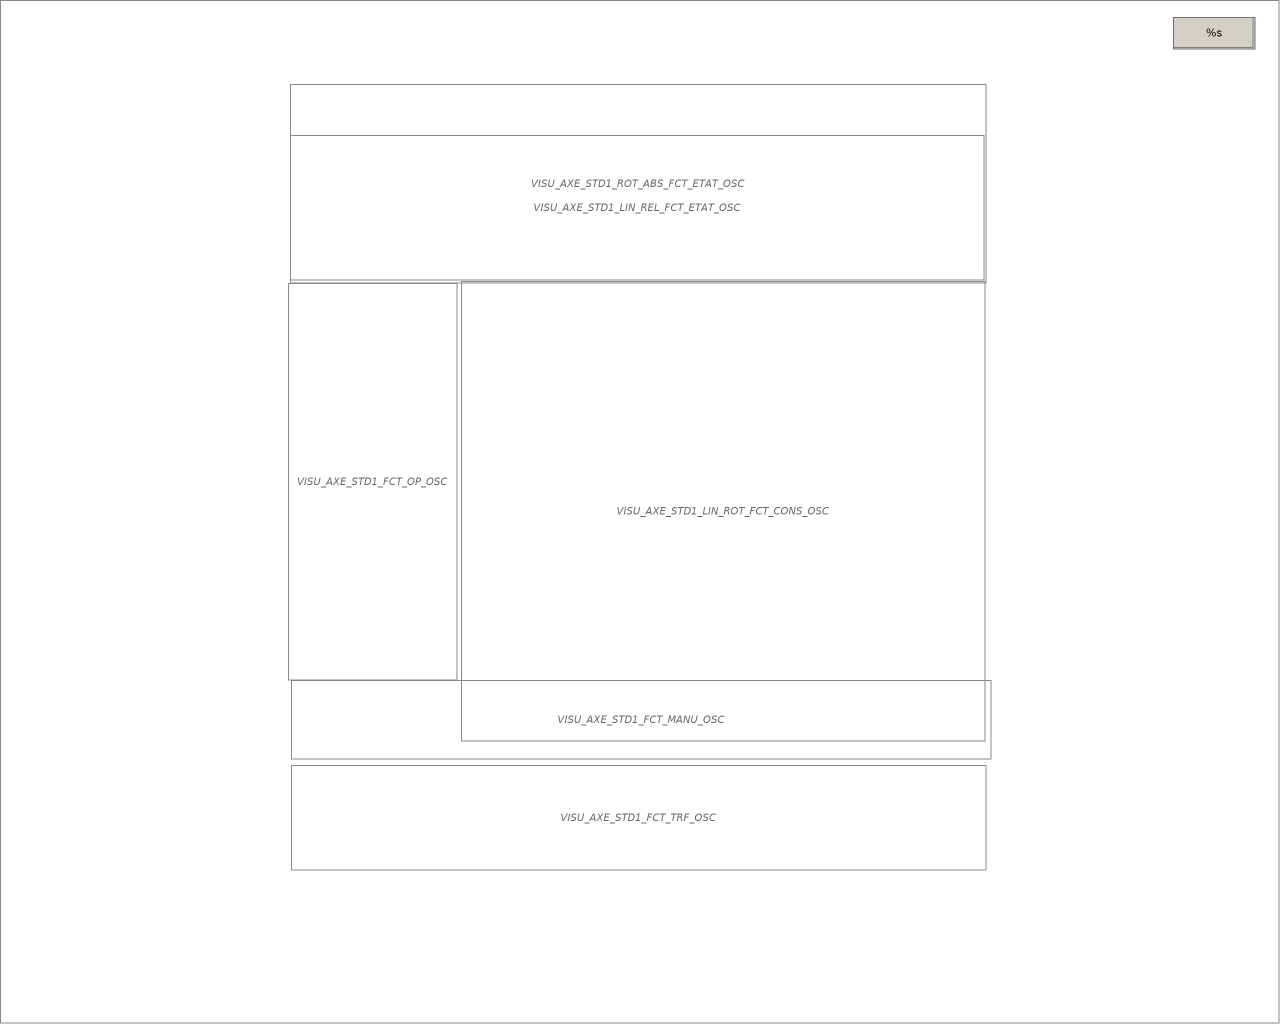
VISUALIZATION VISU_AXE_STD1_MANU_OSC  // 1280x1024
VAR_IN_OUT
	m_Input_MOTEUR: BLOCK_AXE_STD1_OSCILLANT;
	m_Input_PRG_MOUVEMENT_PS: BLOCK_PRG_MOUVEMENT_PS;
END_VAR
VAR_INPUT
	m_Input_ID_NOM_XML : INT;
	m_Input_INDEX_MOTEUR : INT;
	m_Input_Ref_Trf:	USINT;
END_VAR
    Frame (290,84 696x199), invisible if: NOT m_Input_PRG_MOUVEMENT_PS.CONF_ROT_ABS[m_Input_INDEX_MOTEUR]
        shows VISU_AXE_STD1_ROT_ABS_FCT_ETAT_OSC(m_Input_MOTEUR := m_Input_MOTEUR, m_Input_PRG_MOUVEMENT_PS := m_Input_PRG_MOUVEMENT_PS, m_Input_ID_NOM_XML := m_Input_ID_NOM_XML, m_Input_INDEX_MOTEUR := m_Input_INDEX_MOTEUR)
        p625233746: m_Input_MOTEUR
        p171577005: m_Input_PRG_MOUVEMENT_PS
        p3150284580: m_Input_ID_NOM_XML
        p114361821: m_Input_INDEX_MOTEUR
    Button (1173,17 82x32), "%s", text list: 'TextList_Basiques', text index: 8
        OnMouseClick: change screen: Previous 
        OnMouseClick: execute { .VISU_INDEX_MANU := 0; }
    Frame (290,135 694x145), invisible if: NOT m_Input_PRG_MOUVEMENT_PS.CONF_LIN_REL[m_Input_INDEX_MOTEUR]
        shows VISU_AXE_STD1_LIN_REL_FCT_ETAT_OSC(m_Input_MOTEUR := m_Input_MOTEUR, m_Input_PRG_MOUVEMENT_PS := m_Input_PRG_MOUVEMENT_PS, m_Input_ID_NOM_XML := m_Input_ID_NOM_XML)
        p625233746: m_Input_MOTEUR
        p171577005: m_Input_PRG_MOUVEMENT_PS
        p3150284580: m_Input_ID_NOM_XML
    Frame (288,283 169x397)
        shows VISU_AXE_STD1_FCT_OP_OSC(m_Input_MOTEUR := m_Input_MOTEUR, m_Input_PRG_MOUVEMENT_PS := m_Input_PRG_MOUVEMENT_PS, m_Input_INDEX_MOTEUR := m_Input_INDEX_MOTEUR)
        p625233746: m_Input_MOTEUR
        p171577005: m_Input_PRG_MOUVEMENT_PS
        p114361821: m_Input_INDEX_MOTEUR
    Frame (461,281 524x460), invisible if: NOT m_Input_PRG_MOUVEMENT_PS.CONF_LIN_REL[m_Input_INDEX_MOTEUR] AND NOT m_Input_PRG_MOUVEMENT_PS.CONF_ROT_ABS[m_Input_INDEX_MOTEUR]
        shows VISU_AXE_STD1_LIN_ROT_FCT_CONS_OSC(m_Input_MOTEUR := m_Input_MOTEUR, m_Input_PRG_MOUVEMENT_PS := m_Input_PRG_MOUVEMENT_PS, m_Input_INDEX_MOTEUR := m_Input_INDEX_MOTEUR)
        p625233746: m_Input_MOTEUR
        p171577005: m_Input_PRG_MOUVEMENT_PS
        p114361821: m_Input_INDEX_MOTEUR
    Frame (291,680 700x79)
        shows VISU_AXE_STD1_FCT_MANU_OSC(m_Input_MOTEUR := m_Input_MOTEUR, m_Input_PRG_MOUVEMENT_PS := m_Input_PRG_MOUVEMENT_PS, m_Input_INDEX_MOTEUR := m_Input_INDEX_MOTEUR)
        p625233746: m_Input_MOTEUR
        p171577005: m_Input_PRG_MOUVEMENT_PS
        p114361821: m_Input_INDEX_MOTEUR
    Frame (291,765 695x105), invisible if: NOT m_Input_PRG_MOUVEMENT_PS.CONF_TRF[m_Input_INDEX_MOTEUR]
        shows VISU_AXE_STD1_FCT_TRF_OSC(m_Input_MOTEUR := m_Input_MOTEUR, m_Input_PRG_MOUVEMENT_PS := m_Input_PRG_MOUVEMENT_PS, m_Input_INDEX_MOTEUR := m_Input_INDEX_MOTEUR, m_Input_Ref_Trf := m_Input_REF_TRF)
        p625233746: m_Input_MOTEUR
        p171577005: m_Input_PRG_MOUVEMENT_PS
        p114361821: m_Input_INDEX_MOTEUR
        p3023144840: m_Input_REF_TRF
END_VISUALIZATION

(* stored: Version 1.1.0.1, ProductVersion 3.1.4024.10
   Visu VISU_AXE_STD1_MANU_OSC: Id {8d001aba-c871-4aca-94b5-502b472de006} *)
